FUNCTION_BLOCK KeyValueCollectionChangedEventHandler EXTENDS KeyValueCollectionEventHandler

METHOD PUBLIC HandleEvent
VAR_INPUT
	Event : I_Event;
END_VAR
VAR
	changedEvent : I_KeyValueCollectionChangedEvent;
END_VAR
IF __QUERYINTERFACE(Event, changedEvent) THEN
	_eventReceived := TRUE;
	fromExpected := changedEvent.Target = expectedOriginator;
END_IF
END_METHOD

END_FUNCTION_BLOCK

(* stored: Version 1.1.0.1, ProductVersion 3.1.4024.12
   POU KeyValueCollectionChangedEventHandler: Id {00f710aa-2192-0783-217e-a3436cd93408}, SpecialFunc None
   Method HandleEvent: Id {ad60e439-042d-0929-20db-6b7dcab5f136} *)
